{attribute 'GeneratedUsingTerminal: EM7004-0000-9995'}
{attribute addProperty BoxType "EM7004-0000-9995"}
{attribute addProperty Id "InputAT %I*ARRAY[0..15] OF BOOL16"}
{attribute addProperty CRC "2621435360"}
{attribute addProperty Size "16"}
TYPE Digital_BD004D6F :
STRUCT
	{attribute addProperty Name "Input"}
	Input AT %I* : ARRAY[0..15] OF BOOL;
END_STRUCT
END_TYPE

(* stored: Version 1.2.0.0, ProductVersion 3.1.4024.9
   DUT Digital_BD004D6F: Id {b573b471-d002-4176-b82b-ec823c4e2b44} *)
